SUBAPPLICATION Uebung_020c2 (* DigitalInput_I1 auf DigitalOutput_Q1; E_TON Einschaltverzögert; Zeit eingeben und speichern. *)
  (* Standard: 61499-2 *)
  (* Version 1.0, 2023-10-23, franz *)
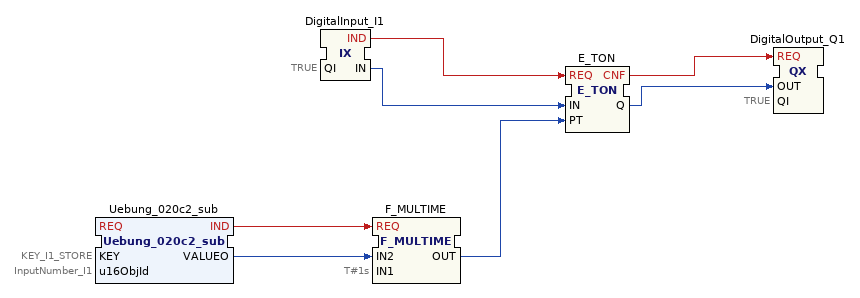
  FBS
    DigitalOutput_Q1 : QX(QI := TRUE);
    DigitalInput_I1 : IX(QI := TRUE);
    E_TON : E_TON;
    F_MULTIME : F_MULTIME(IN1 := T#1s);
  END_FBS
  SUBAPPS
    Uebung_020c2_sub : Uebung_020c2_sub(KEY := KEY_I1_STORE, u16ObjId := InputNumber_I1);
  END_SUBAPPS
  EVENT_CONNECTIONS
    DigitalInput_I1.IND TO E_TON.REQ;
    E_TON.CNF TO DigitalOutput_Q1.REQ;
    Uebung_020c2_sub.IND TO F_MULTIME.REQ;
  END_CONNECTIONS
  DATA_CONNECTIONS
    DigitalInput_I1.IN TO E_TON.IN;
    E_TON.Q TO DigitalOutput_Q1.OUT;
    F_MULTIME.OUT TO E_TON.PT;
    Uebung_020c2_sub.VALUEO TO F_MULTIME.IN2;
  END_CONNECTIONS
END_SUBAPPLICATION
